FUNCTION_BLOCK DoorSensor (* Basic Function Block Type *)
  (* Standard: 61499-2 *)
  (* Version 0.0, 6/3/2016, Andrei, nxtControl GmbH, Template *)
  PACKAGE Main;
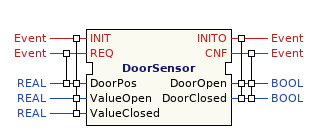
  EVENT_INPUT
    INIT WITH DoorPos, ValueOpen, ValueClosed; (* Initialization Request *)
    REQ WITH DoorPos; (* Normal Execution Request *)
  END_EVENT
  EVENT_OUTPUT
    INITO WITH DoorOpen, DoorClosed; (* Initialization Confirm *)
    CNF WITH DoorOpen, DoorClosed; (* Execution Confirmation *)
  END_EVENT
  VAR_INPUT
    DoorPos : REAL; (* Input event qualifier *)
    ValueOpen : REAL;
    ValueClosed : REAL;
  END_VAR
  VAR_OUTPUT
    DoorOpen : BOOL; (* Output event qualifier *)
    DoorClosed : BOOL;
  END_VAR
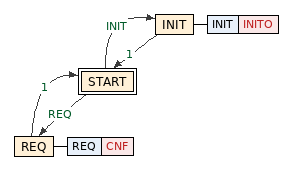
  EC_STATES
    START; (* Initial State *)
    INIT : INIT -> INITO; (* Initialization *)
    REQ : REQ -> CNF; (* Normal execution *)
  END_STATES
  EC_TRANSITIONS
    START TO INIT := INIT;
    INIT TO START := 1;
    START TO REQ := REQ;
    REQ TO START := 1;
  END_TRANSITIONS
  ALGORITHM INIT IN ST: (* Initialization algorithm *)
;
  END_ALGORITHM
  ALGORITHM REQ IN ST: (* Normally executed algorithm *)
IF DoorPos > ValueOpen THEN
	DoorOpen := TRUE;
	DoorClosed := FALSE;
ELSIF DoorPos < ValueClosed THEN
	DoorOpen := FALSE;
	DoorClosed := TRUE;
ELSE
	DoorOpen := FALSE;
	DoorClosed := FALSE;
END_IF;
  END_ALGORITHM
END_FUNCTION_BLOCK
